Fanuc KAREL source: kt00089.compact.KL

PROGRAM KT00089
%STACKSIZE=65535
%PRIORITY=65535
%NOLOCKGROUP
VAR
H1 : ARRAY[2] OF SHORT
I2 : INTEGER
OUT : INTEGER
BEGIN
H1[1]=2
I2=3
OUT=(H1[1] * I2)
END KT00089
